# EPICS autosave request: measCompApp/Db/USB1808_settings.req
file "measCompBinaryDir_settings.req",    P=$(P), R=Bd1
file "measCompBinaryDir_settings.req",    P=$(P), R=Bd2
file "measCompBinaryDir_settings.req",    P=$(P), R=Bd3
file "measCompBinaryDir_settings.req",    P=$(P), R=Bd4
file "measCompPulseGen_settings.req",     P=$(P), R=PulseGen1
file "measCompPulseGen_settings.req",     P=$(P), R=PulseGen2
file "measCompAnalogInMode_settings.req", P=$(P), R=AiMode
file "measCompAnalogIn_settings.req",     P=$(P), R=Ai1
file "measCompAnalogIn_settings.req",     P=$(P), R=Ai2
file "measCompAnalogIn_settings.req",     P=$(P), R=Ai3
file "measCompAnalogIn_settings.req",     P=$(P), R=Ai4
file "measCompAnalogIn_settings.req",     P=$(P), R=Ai5
file "measCompAnalogIn_settings.req",     P=$(P), R=Ai6
file "measCompAnalogIn_settings.req",     P=$(P), R=Ai7
file "measCompAnalogIn_settings.req",     P=$(P), R=Ai8
file "measCompAnalogOut_settings.req",    P=$(P), R=Ao1
file "measCompAnalogOut_settings.req",    P=$(P), R=Ao2
file "measCompWaveformDig_settings.req",  P=$(P), R=WaveDig
file "measCompWaveformGen_settings.req",  P=$(P), R=WaveGen
file "measCompWaveformGenN_settings.req", P=$(P), R=WaveGen1
file "measCompWaveformGenN_settings.req", P=$(P), R=WaveGen2
file "measCompTrigger_settings.req",      P=$(P), R=Trig
